// TIA Portal V16 export
// export: Created 2025-12-18T09:29:14.6700175Z, ExportSetting WithDefaults, DisplayName Totally Integrated Automation Portal, DisplayVersion V16, DisplayName TIA Portal Version Control Interface, DisplayVersion V16, DisplayName TIA Portal Openness, DisplayVersion V16, DisplayName STEP 7 Professional, DisplayVersion V16, DisplayName STEP 7 Safety, DisplayVersion V16, DisplayName WinCC Advanced, DisplayVersion V16
FUNCTION_BLOCK "Supply Conveyor"   // FB6, LAD
{ S7_Optimized_Access := 'TRUE' }
VERSION : 0.1
// stored: AutoNumber true, IsIECCheckEnabled false, IsRetainMemResEnabled false, MemoryReserve 100, SetENOAutomatically false, UDAEnableTagReadback false
   VAR
      xMaterialOnConveyor : Bool;
      xEdgeMemory1 { ExternalAccessible := 'False'; ExternalVisible := 'False'; ExternalWritable := 'False'} : Bool;
      xEdgeMemory2 { ExternalAccessible := 'False'; ExternalVisible := 'False'; ExternalWritable := 'False'} : Bool := false;
      xEdgeMemory3 { ExternalAccessible := 'False'; ExternalVisible := 'False'; ExternalWritable := 'False'} : Bool := false;
   END_VAR
   VAR_TEMP   // added for the SCL form of the ladder/FBD networks
      _w1 : Bool;
      _w2 : Bool;
   END_VAR
BEGIN

REGION Network 1
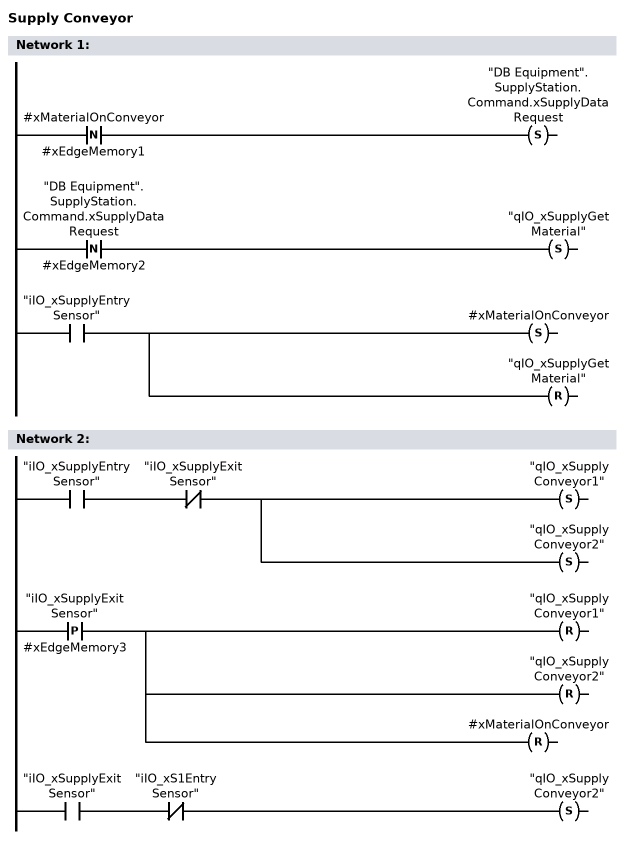
   RUNG wire#powerrail
      N_Contact(operand := #xMaterialOnConveyor, bit := #xEdgeMemory1)
      S_Coil( "DB Equipment".SupplyStation.Command.xSupplyDataRequest )
   END_RUNG
   RUNG wire#powerrail
      N_Contact(operand := "DB Equipment".SupplyStation.Command.xSupplyDataRequest, bit := #xEdgeMemory2)
      S_Coil( "qIO_xSupplyGetMaterial" )
   END_RUNG
   RUNG wire#powerrail
      Contact( "iIO_xSupplyEntrySensor" )
      wire#w1
      S_Coil( #xMaterialOnConveyor )
   END_RUNG
   RUNG wire#w1
      R_Coil( "qIO_xSupplyGetMaterial" )
   END_RUNG
   // the same network as SCL:
   #_w1 := NOT #xMaterialOnConveyor AND #xEdgeMemory1;   // falling edge of #xMaterialOnConveyor
   #xEdgeMemory1 := #xMaterialOnConveyor;
   IF #_w1 THEN "DB Equipment".SupplyStation.Command.xSupplyDataRequest := TRUE; END_IF;
   #_w2 := NOT "DB Equipment".SupplyStation.Command.xSupplyDataRequest AND #xEdgeMemory2;   // falling edge of "DB Equipment".SupplyStation.Command.xSupplyDataRequest
   #xEdgeMemory2 := "DB Equipment".SupplyStation.Command.xSupplyDataRequest;
   IF #_w2 THEN "qIO_xSupplyGetMaterial" := TRUE; END_IF;
   IF "iIO_xSupplyEntrySensor" THEN
       #xMaterialOnConveyor := TRUE;
       "qIO_xSupplyGetMaterial" := FALSE;
   END_IF;
END_REGION

REGION Network 2
   RUNG wire#powerrail
      Contact( "iIO_xSupplyEntrySensor" )
      I_Contact( "iIO_xSupplyExitSensor" )
      wire#w1
      S_Coil( "qIO_xSupplyConveyor1" )
   END_RUNG
   RUNG wire#w1
      S_Coil( "qIO_xSupplyConveyor2" )
   END_RUNG
   RUNG wire#powerrail
      P_Contact(operand := "iIO_xSupplyExitSensor", bit := #xEdgeMemory3)
      wire#w2
      R_Coil( "qIO_xSupplyConveyor1" )
   END_RUNG
   RUNG wire#w2
      R_Coil( "qIO_xSupplyConveyor2" )
   END_RUNG
   RUNG wire#w2
      R_Coil( #xMaterialOnConveyor )
   END_RUNG
   RUNG wire#powerrail
      Contact( "iIO_xSupplyExitSensor" )
      I_Contact( "iIO_xS1EntrySensor" )
      S_Coil( "qIO_xSupplyConveyor2" )
   END_RUNG
   // the same network as SCL:
   IF "iIO_xSupplyEntrySensor" AND NOT "iIO_xSupplyExitSensor" THEN
       "qIO_xSupplyConveyor1" := TRUE;
       "qIO_xSupplyConveyor2" := TRUE;
   END_IF;
   #_w1 := "iIO_xSupplyExitSensor" AND NOT #xEdgeMemory3;   // rising edge of "iIO_xSupplyExitSensor"
   #xEdgeMemory3 := "iIO_xSupplyExitSensor";
   IF #_w1 THEN
       "qIO_xSupplyConveyor1" := FALSE;
       "qIO_xSupplyConveyor2" := FALSE;
       #xMaterialOnConveyor := FALSE;
   END_IF;
   IF "iIO_xSupplyExitSensor" AND NOT "iIO_xS1EntrySensor" THEN "qIO_xSupplyConveyor2" := TRUE; END_IF;
END_REGION
END_FUNCTION_BLOCK
